PROGRAM MAIN
VAR
	i,j : T_Position;
	Comp : T_Comparison;
	bAdd, bRemove, bClear : BOOL;
	fbSet : FB_Tree_Set;
	fbMap : FB_Tree_Map;
	Data : ARRAY[0..10] OF INT := [1,2,3,4,5,6,7,8,9,10];
END_VAR

Comp := F_Compare_Any(i,j);

IF bAdd THEN
	bAdd := FALSE;
	FOR i := 0 TO 3 DO fbSet.Insert(i); END_FOR
	END_IF

IF bRemove THEN 
	bRemove := FALSE;
	fbSet.Remove(j);
	END_IF
	
IF bClear THEN 
	bClear := FALSE;
	fbSet.Clear();
	END_IF

END_PROGRAM

(* stored: Version 1.1.0.1, ProductVersion 3.1.4024.4
   POU MAIN: Id {17732e83-93d3-4e32-896f-74d26e2dd9ab}, SpecialFunc None *)
